// TIA Portal V17 export
// export: Created 2025-03-05T08:02:49.8603278Z, ExportSetting WithDefaults, DisplayName Totally Integrated Automation Portal, DisplayVersion V17 Update 8, DisplayName TIA Portal Openness, DisplayVersion V17 Update 8, DisplayName TIA Portal Version Control Interface, DisplayVersion V17, DisplayName SINAMICS Startdrive Advanced, DisplayVersion V17 SP2, DisplayName SINAMICS Startdrive G110M, G120, G120C, G120D, G120P, G115D, DisplayVersion V17 SP2, DisplayName SINAMICS Startdrive G130, G150, S120, S150, SINAMICS MV, S210, DisplayVersion V17 SP2, DisplayName STEP 7 Professional, DisplayVersion V17 Update 8, DisplayName SINUMERIK ONE STEP 7 Toolbox, DisplayVersion V17 Update 12, DisplayName SINUMERIK 840D sl STEP 7 Toolbox, DisplayVersion V17 Update 12, DisplayName STEP 7 Safety, DisplayVersion V17 Update 6, DisplayName WinCC Advanced, DisplayVersion V17 Update 8
DATA_BLOCK "DB2103_ELECTRICAL_CABINET"   // DB2103
{ S7_Optimized_Access := 'FALSE'; DB_Accessible_From_OPC_UA := 'FALSE' }
AUTHOR : ETXETAR
VERSION : 1.0
// stored: AutoNumber false, DBAccessibleFromOPCUA false, DBAccessibleFromWebserver true, IsOnlyStoredInLoadMemory false, IsWriteProtectedInAS false
   VAR RETAIN
      INPUT_230_VAC_BREAKER : Bool;   // MAIN CABINET CIRCUIT BREAKER TRIPPED / INPUT 230 VAC CABINET CIRCUIT BREAKER TRIPPED
      INPUT_AIR_UNIT_1_BREAKER : Bool;   // AIR UNIT BREAKER - STOP END OF CYCLE / INPUT AIR UNIT 1 CRICUIT BREAKER TRIPPED
      INPUT_AIR_UNIT_2_BREAKER : Bool;   // AIR UNIT BREAKER - STOP END OF CYCLE / INPUT AIR UNIT 2 CIRCUIT BREAKER TRIPPED
      INPUT_24VDC_BREAKER_1 : Bool;   // CIRCUIT BREAKER 24 V DC / INPUT 24 VDC CIRCUIT BREAKER TRIPPED 1
      INPUT_24VDC_BREAKER_2 : Bool;   // CIRCUIT BREAKER 24 V DC / INPUT 24 VDC CIRCUIT BREAKER TRIPPED 2
      INPUT_FC35_1_BREAKER : Bool;   // INPUT BREAKER 3004 / INPUT FC35.1 CIRCUIT BREAKER TRIPPED
      INPUT_FC35_2_BREAKER : Bool;   // INPUT FC35.2 CIRCUIT BREAKER TRIPPED
      INPUT_FC35_3_BREAKER : Bool;   // INPUT FC35.3 CIRCUIT BREAKER TRIPPED
      INPUT_SINAMICS_BREAKER : Bool;   // SINAMICS CIRCUIT BREAKER TRIPPED INPUT / INPUT SINAMICS CIRCUIT BREAKER TRIPPED
      "INPUT_110/120/220/230VAC_BREAKER" : Bool;   // CIRCUIT BREAKER F1 - F4 / INPUT 110/120/220/230VAC CIRCUIT BREAKER TRIPPED
      INPUT_SINAMICS_BREAKER_1 : Bool;   // INPUT SINAMICS CIRCUIT BREAKER TRIPPED
      INPUT_CAB_LIGHT_BREAKER : Bool;   // CIRCUIT BREAKER CABINET LIGHTING / INPUT CABINET LIGHT CIRCUIT BREAKER TRIPPED
      INPUT_SENTRON_PAC_BREAKER : Bool;   // INPUT BREAKER SENTRON PAC3200 / INPUT SENTRON PAC CIRCUIT BREAKER TRIPPED
      INPUT_JIB_CRANE_BREAKER : Bool;   // CIRCUIT BREAKER JIB CRANE / INPUT JIB CRANE CIRCUIT BREAKER TRIPPED
      INPUT_MAIN_SWITCH : Bool;   // ELECTRICAL CABINET MAIN SWITCH INPUT / INPUT MAIN SWITCH
      INPUT_PANEL_TEMPERATURE : Bool;   // PANEL TEMPERATURE STOP END OF CYCLE / INPUT PANEL TEMPERATURE
      INPUT_AIR_UNIT_1 : Bool;   // AIR UNIT OK - STOP END OF CYCLE / INPUT AIR UNIT 1
      INPUT_AIR_UNIT_2 : Bool;   // AIR UNIT OK - STOP END OF CYCLE / INPUT AIR UNIT 2
      INPUT_OVER_VOLTAGE : Bool;   // INPUT OVER VOLTAGE
      INPUT_POWER_SUPPLY : Bool;   // FAULT POWER SUPPLY / INPUT POWER SUPPLY
      INPUT_PS_24V_NOT_READY_DEV_1 : Bool;   // INPUT POWER SUPPLY 24V NOT READY DEVICE 1
      INPUT_PS_24V_NOT_READY_DEV_2 : Bool;   // INPUT POWER SUPPLY 24V NOT READY DEVICE 2
      INPUT_PS_24V_NOT_READY_DEV_3 : Bool;   // INPUT POWER SUPPLY 24V NOT READY DEVICE 3
      INPUT_PS_24V_NOT_READY_DEV_4 : Bool;   // INPUT POWER SUPPLY 24V NOT READY DEVICE 4
      INPUT_PS_24V_NOT_READY_DEV_5 : Bool;   // INPUT POWER SUPPLY 24V NOT READY DEVICE 5
      INPUT_PS_24V_NOT_READY_DEV_6 : Bool;   // INPUT POWER SUPPLY 24V NOT READY DEVICE 6
      INPUT_BATTERY_OK_SITOP_UPS500S : Bool;   // INPUT BATTERY OK SITOP UPS500S
      INPUT_BATTERY_ALARM_SITOP_UPS500S : Bool;   // INPUT BATTERY ALARM SITOP UPS500S
      INPUT_ETHERNET_SWITCH_1 : Bool;   // INPUT SWITCH ETHERNET SWITCH 1 FAULT / INPUT ETHERNET SWITCH 1
      INPUT_ETHERNET_SWITCH_2 : Bool;   // INPUT SWITCH ETHERNET SWITCH 2 FAULT / INPUT ETHERNET SWITCH 2
      INPUT_ETHERNET_SWITCH_3 : Bool;   // INPUT SWITCH ETHERNET SWITCH 3 FAULT / INPUT ETHERNET SWITCH 3
      INPUT_ETHERNET_SWITCH_4 : Bool;   // INPUT ETHERNET SWITCH 4
      INPUT_ELEC_CAB_DOOR_OPEN : Bool;   // INPUT ELECTRICAL CABINET DOOR OPENED / INPUT ELECTRICAL CABINET DOOR OPEN
      INPUT_BATTERY_85_SITOP_UPS500S : Bool;   // INPUT BATTERY 85% SITOP UPS500S
      INPUT_PS_24V_BREAKER_DEV_1 : Bool;   // POWER SUPPLY 24V CIRCUIT BREAKER TRIPPED DEVICE 1 INPUT (WITHOUT FB) / INPUT POWER SUPPLY 24V CIRCUIT BREAKER TRIPPED DEVICE 1
      INPUT_PS_24V_BREAKER_DEV_2 : Bool;   // POWER SUPPLY 24V CIRCUIT BREAKER TRIPPED DEVICE 2 INPUT (WITHOUT FB) / INPUT POWER SUPPLY 24V CIRCUIT BREAKER TRIPPED DEVICE 2
      INPUT_PS_24V_BREAKER_DEV_3 : Bool;   // POWER SUPPLY 24V CIRCUIT BREAKER TRIPPED DEVICE 3 INPUT (WITHOUT FB) / INPUT POWER SUPPLY 24V CIRCUIT BREAKER TRIPPED DEVICE 3
      INPUT_PS_24V_BREAKER_DEV_4 : Bool;   // POWER SUPPLY 24V CIRCUIT BREAKER TRIPPED DEVICE 4 INPUT (WITHOUT FB) / INPUT POWER SUPPLY 24V CIRCUIT BREAKER TRIPPED DEVICE 4
      INPUT_LASER_BREAKER_U01 : Bool;   // INPUT LASER SOURCE UNIT 01 CIRCUIT BREAKER TRIPPED
      INPUT_LASER_BREAKER_U02 : Bool;   // INPUT LASER SOURCE UNIT 02 CIRCUIT BREAKER TRIPPED
      INPUT_OERLIKON_BREAKER_U01 : Bool;   // INPUT OERLIKON SOURCE UNIT 01 CIRCUIT BREAKER TRIPPED
      INPUT_OERLIKON_BREAKER_U02 : Bool;   // INPUT OERLIKON SOURCE UNIT 02 CIRCUIT BREAKER TRIPPED
      INPUT_HEATER_BREAKER : Bool;   // INPUT HEATER CIRCUIT BREAKER TRIPPED
      INPUT_AXIS_Z11_BREAKER_1 : Bool;   // INPUT AXIS Z11 CIRCUIT BREAKER 1 TRIPPED
      INPUT_AXIS_Z11_BREAKER_2 : Bool;   // INPUT AXIS Z11 CIRCUIT BREAKER 2 TRIPPED
      INPUT_STIRRER_BREAKER : Bool;   // INPUT STIRRER CIRCUIT BREAKER 2 TRIPPED
      INPUT_CHILLER_BREAKER_1 : Bool;   // INPUT CHILLER CIRCUIT BREAKER 2 TRIPPED
      INPUT_HOPPERS_BREAKER : Bool;   // INPUT HOPPERS CIRCUIT BREAKER 2 TRIPPED
      INPUT_AXIS_Z21_BREAKER_1 : Bool;   // INPUT AXIS Z21 CIRCUIT BREAKER 1 TRIPPED
      INPUT_AXIS_Z21_BREAKER_2 : Bool;   // INPUT AXIS Z21 CIRCUIT BREAKER 2 TRIPPED
      "230_VAC_BREAKER_TRIPPED_ALARM" : Bool;   // MAIN CIRCUIT BREAKER FAULT / 230 VAC BREAKER TRIPPED ALARM
      INPUT_PILZ_ESTOP_OK : Bool;   // INPUT PILZ EMERGENCY STOP OK
      AIR_UNIT_1_BREAKER_TRIPPED_ALARM : Bool;   // AIR UNIT CIRCUIT BREAKER FAULT / AIR UNIT 1 CIRCUIT BREAKER TRIPPED ALARM
      AIR_UNIT_2_BREAKER_TRIPPED_ALARM : Bool;   // AIR UNIT CIRCUIT BREAKER FAULT / AIR UNIT 2 CIRCUIT BREAKER TRIPPED ALARM
      "24VDC_BREAKER_TRIPPED_ALARM_1" : Bool;   // CIRCUIT BREAKER 24 V DC FAULT / 24 VDC CIRCUIT BREAKER TRIPPED 1 ALARM
      "24VDC_BREAKER_TRIPPED_ALARM_2" : Bool;   // AUXILIAR CIRCUIT BRAKER 24 VDC FAULT / 24 VDC CIRCUIT BREAKER TRIPPED 2 ALARM
      FC35_1_BREAKER_TRIPPED_ALARM : Bool;   // BREAKER QF3004 FAULT / FC35.1 CIRCUIT BREAKER TRIPPED ALARM
      FC35_2_BREAKER_TRIPPED_ALARM : Bool;   // BREAKER QF3004 FAULT / FC35.2 CIRCUIT BREAKER TRIPPED ALARM
      FC35_3_BREAKER_TRIPPED_ALARM : Bool;   // BREAKER QF3004 FAULT / FC35.3 CIRCUIT BREAKER TRIPPED ALARM
      SINAMICS_BREAKER_TRIPPED_ALARM : Bool;   // SINAMICS CIRCUIT BREAKER TRIPPED FAULT / SINAMICS CIRCUIT BREAKER TRIPPED ALARM
      MAIN_SWITCH_ALARM : Bool;   // MAIN SWITCH OFF FAULT / MAIN SWITCH ALARM
      PANEL_TEMPERATURE_ALARM : Bool;   // PANEL TEMPERATURE NOT OK - STOP END OF CYCLE / PANEL TEMPERATURE ALARM
      AIR_UNIT_ALARM_1 : Bool;   // AIR UNIT NOT OK - STOP END OF CYCLE / AIR UNIT 1 ALARM
      AIR_UNIT_ALARM_2 : Bool;   // AIR UNIT NOT OK - STOP END OF CYCLE / AIR UNIT 2 ALARM
      OVER_VOLTAGE_ALARM : Bool;   // OVER VOLTAGE FAULT / OVER VOLTAGE ALARM
      POWER_SUPPLY_ALARM : Bool;   // POWER SUPPLY FAULT / POWER SUPPLY ALARM
      PS_24V_NOT_READY_DEV_ALARM_1 : Bool;   // POWER SUPPLY 24V NOT READY DEVICE 1 ALARM
      PS_24V_NOT_READY_DEV_ALARM_2 : Bool;   // POWER SUPPLY 24V NOT READY DEVICE 2 ALARM
      PS_24V_NOT_READY_DEV_ALARM_3 : Bool;   // POWER SUPPLY 24V NOT READY DEVICE 3 ALARM
      PS_24V_NOT_READY_DEV_ALARM_4 : Bool;   // POWER SUPPLY 24V NOT READY DEVICE 4 ALARM
      PS_24V_NOT_READY_DEV_ALARM_5 : Bool;   // POWER SUPPLY 24V NOT READY DEVICE 5 ALARM
      PS_24V_NOT_READY_DEV_ALARM_6 : Bool;   // POWER SUPPLY 24V NOT READY DEVICE 6 ALARM
      BATTERY_OK_SITOP_UPS500S_ALARM : Bool;   // SITOP UPS500S BATTERY NOT OK ALARM / BATTERY OK SITOP UPS500S ALARM
      BATTERY_ALARM_SITOP_UPS500S : Bool;   // SITOP UPS500S BATTERY LOW LEVEL ALARM / BATTERY ALARM SITOP UPS500S ALARM
      ETHERNET_SWITCH_1_ALARM : Bool;   // SWITCH SCALANCE X108 FAIL / ETHERNET SWITCH 1 ALARM
      ETHERNET_SWITCH_2_ALARM : Bool;   // ETHERNET SWITCH 2 ALARM
      ETHERNET_SWITCH_3_ALARM : Bool;   // ETHERNET SWITCH 3 ALARM
      ETHERNET_SWITCH_4_ALARM : Bool;   // ETHERNET SWITCH 4 ALARM
      PS_24V_BREAKER_TRIPPED_ALARM_DEV_1 : Bool;   // DIAGNOSIS 24V MODULE CIRCUIT BREAKER 1 TRIPPED / POWER SUPPLY 24V CIRCUIT BREAKER TRIPPED DEVICE 1 ALARM
      PS_24V_BREAKER_TRIPPED_ALARM_DEV_2 : Bool;   // DIAGNOSIS 24V MODULE CIRCUIT BREAKER 2 TRIPPED / POWER SUPPLY 24V CIRCUIT BREAKER TRIPPED DEVICE 2 ALARM
      PS_24V_BREAKER_TRIPPED_ALARM_DEV_3 : Bool;   // DIAGNOSIS 24V MODULE CIRCUIT BREAKER 3 TRIPPED / POWER SUPPLY 24V CIRCUIT BREAKER TRIPPED DEVICE 3 ALARM
      PS_24V_BREAKER_TRIPPED_ALARM_DEV_4 : Bool;   // DIAGNOSIS 24V MODULE CIRCUIT BREAKER 4 TRIPPED / POWER SUPPLY 24V CIRCUIT BREAKER TRIPPED DEVICE 4 ALARM
      SINAMICS_BREAKER_ALARM : Bool;   // SINAMICS CIRCUIT BREAKER TRIPPED ALARM
      LASER_BREAKER_U01_ALARM : Bool;   // ALARM LASER SOURCE UNIT 01 CIRCUIT BREAKER TRIPPED
      LASER_BREAKER_U02_ALARM : Bool;   // ALARM LASER SOURCE UNIT 02 CIRCUIT BREAKER TRIPPED
      OERLIKON_BREAKER_U01_ALARM : Bool;   // ALARM OERLIKON SOURCE UNIT 01 CIRCUIT BREAKER TRIPPED
      OERLIKON_BREAKER_U02_ALARM : Bool;   // ALARM OERLIKON SOURCE UNIT 02 CIRCUIT BREAKER TRIPPED
      HEATER_BREAKER_ALARM : Bool;   // ALARM HEATER CIRCUIT BREAKER TRIPPED
      AXIS_Z11_BREAKER_1_ALARM : Bool;   // ALARM AXIS Z11 CIRCUIT BREAKER 1 TRIPPED
      AXIS_Z11_BREAKER_2_ALARM : Bool;   // ALARM AXIS Z11 CIRCUIT BREAKER 2 TRIPPED
      STIRRER_BREAKER_ALARM : Bool;   // ALARM STIRRER CIRCUIT BREAKER TRIPPED
      CHILLER_BREAKER_ALARM : Bool;   // ALARM CHILLER CIRCUIT BREAKER TRIPPED
      HOPPERS_BREAKER_ALARM : Bool;   // ALARM HOPPERS CIRCUIT BREAKER TRIPPED
      AXIS_Z21_BREAKER_1_ALARM : Bool;   // ALARM AXIS Z21 CIRCUIT BREAKER 1 TRIPPED
      AXIS_Z21_BREAKER_2_ALARM : Bool;   // ALARM AXIS Z21 CIRCUIT BREAKER 2 TRIPPED
      "110/120/220/230VAC_BREAKER_TRIPPED_WARNING" : Bool;   // BREAKER 120VA TRIPPED / 110/120/220/230VAC CIRCUIT BREAKER TRIPPED WARNING
      CAB_LIGHT_BREAKER_TRIPPED_WARNING : Bool;   // CIRCUIT BREAKER CABINET LIGHTING WARNING / CABINET LIGHT CIRCUIT BREAKER TRIPPED WARNING
      SENTRON_PAC_BREAKER_TRIPPED_WARNING : Bool;   // CIRCUIT BREAKER SENTRON PACK3200 TRIPPED / SENTRON PAC CIRCUIT BREAKER TRIPPED WARNING
      JIB_CRANE_BREAKER_TRIPPED_WARNING : Bool;   // CIRCUIT BREAKER JIB CRANE FAULT / JIB CRANE CIRCUIT BREAKER TRIPPED WARNING
      ELEC_CAB_DOOR_OPEN_WARNING : Bool;   // ELECTRICAL CABINET DOOR OPENED / ELECTRICAL CABINET DOOR OPEN WARNING
      BATTERY_85_SITOP_UPS500S_WARNING : Bool;   // SITOP UPS500S BATTERY 85 WARNING / BATTERY 85% SITOP UPS500S WARNING
      PILZ_ESTOP_OK_ALARM : Bool;   // PILZ EMERGENCY STOP OK ALARM
      ANY_ACTIVE_ALARM : Bool;   // RETURN TO HOME POSITION ALARMS / ANY ACTIVE ALARM
      IS_ALARMS : Bool;   // IMMEDIATE STOP ALARMS
      SEOC_ALARMS : Bool;   // STOP AT END OF CYCLE ALARMS / STOP END OF CYCLE ALARMS
      WARNINGS : Bool;   // WARNING / WARNINGS
      WARNINGS_GONE : Bool;   // WARNING GONE / WARNINGS GONE
      TIMER_SITOP_BATTERY { S7_SetPoint := 'True'} : TON_TIME;   // SITOP BATTERY TIMER
   END_VAR
BEGIN
   TIMER_SITOP_BATTERY.PT := T#5s;
END_DATA_BLOCK
